# EPICS autosave request: mrfApp/Db/evr-template-prescaler-32-bit.inc.req
$(P)$(R)Prescaler@PRESCALER_NUM@.VAL
